(* IEC 61131-3 sources: plc-home-automation/home_automation/lighting_heating_updated/src/lighting, 3 files *)

(* ---- LightingGlobals.st ---- *)
VAR_GLOBAL CONSTANT

    C_DOWNSTAIRS_BATH_MAJOR_LIGHTS_INDEX      : INT := 0;
    C_DOWNSTAIRS_BATH_SHOWER_LIGHTS_INDEX     : INT := 1;
    C_UPSTAIRS_BATH_MAJOR_LIGHTS_INDEX        : INT := 2;
    C_UPSTAIRS_WC_LIGHTS_INDEX                : INT := 3;
    C_UPSTAIRS_BATH_SHOWER_LIGHTS_INDEX       : INT := 4;
    C_HALLWAY_LIGHTS_INDEX                    : INT := 5;
    C_OUTDOOR_LIGHTS_INDEX                    : INT := 6;
    C_HALL_LIGHTS_INDEX                       : INT := 7;
    C_GARAGE_LIGHTS_INDEX                     : INT := 8;
    C_BOILER_LIGHTS_INDEX                     : INT := 9;
    C_MAJOR_STORAGE_LIGHTS_INDEX              : INT := 10;
    C_MINOR_STORAGE_LIGHTS_INDEX              : INT := 11;
    C_GARDEN_BALCONY_LIGHTS_INDEX             : INT := 12;
    C_CHILDRENS_ROOM_2_LIGHTS_INDEX           : INT := 13;
    C_CHILDRENS_ROOM_1_OUTER_LIGHTS_INDEX     : INT := 14;
    C_CHILDRENS_ROOM_1_INNER_LIGHTS_INDEX     : INT := 15;
    C_CHILDRENS_ROOM_3_LIGHTS_INDEX           : INT := 16;
    C_GATE_BALCONY_LIGHTS_INDEX               : INT := 17;
    C_DOWNSTAIRS_BEDROOM_LIGHTS_INDEX         : INT := 18;
    C_KITCHEN_LIGHTS_INDEX                    : INT := 19;
    C_DINING_ROOM_LIGHTS_INDEX                : INT := 20;
    C_LIVING_ROOM_LIGHTS_INDEX                : INT := 21;
    C_TERRACE_LIGHTS_INDEX                    : INT := 22;
//    C_STAIRS_LIGHTS_INDEX               : INT := 23;

    C_LIGHTS_ZONES_COUNT                      : INT := 23;

END_VAR

VAR_GLOBAL

    LIGHTS_INPUTS : ARRAY [0 .. C_LIGHTS_ZONES_COUNT - 1] OF PTR_TO BOOL;
    VIRTUAL_LIGHTS_INPUTS : ARRAY [0 .. C_LIGHTS_ZONES_COUNT - 1] OF PTR_TO BOOL;
    LIGHTS_OUTPUTS : ARRAY [0 .. C_LIGHTS_ZONES_COUNT - 1] OF PTR_TO BOOL;
    LIGHTS_NAMES     : ARRAY [0 .. C_LIGHTS_ZONES_COUNT - 1] OF STRING;

    HALLWAY_LIGHTS_COMBINED_IN : BOOL                      := FALSE;

    VIRTUAL_DOWNSTAIRS_BATH_MAJOR_LIGHTS_IN : BOOL         := FALSE;
    VIRTUAL_DOWNSTAIRS_BATH_SHOWER_LIGHTS_IN : BOOL        := FALSE;
    VIRTUAL_UPSTAIRS_BATH_MAJOR_LIGHTS_IN : BOOL           := FALSE;
    VIRTUAL_UPSTAIRS_WC_LIGHTS_IN : BOOL                   := FALSE;
    VIRTUAL_UPSTAIRS_BATH_SHOWER_LIGHTS_IN : BOOL          := FALSE;
    VIRTUAL_OUTDOOR_LIGHTS_IN : BOOL                       := FALSE;
    VIRTUAL_HALL_LIGHTS_IN : BOOL                          := FALSE;
    VIRTUAL_GARAGE_LIGHTS_IN : BOOL                        := FALSE;
    VIRTUAL_MAJOR_STORAGE_LIGHTS_IN : BOOL                 := FALSE;
    VIRTUAL_MINOR_STORAGE_LIGHTS_IN : BOOL                 := FALSE;
    VIRTUAL_GARDEN_BALCONY_LIGHTS_IN : BOOL                := FALSE;
    VIRTUAL_CHILDRENS_ROOM_2_LIGHTS_IN : BOOL              := FALSE;
    VIRTUAL_CHILDRENS_ROOM_1_OUTER_LIGHTS_IN : BOOL        := FALSE;
    VIRTUAL_CHILDRENS_ROOM_1_INNER_LIGHTS_IN : BOOL        := FALSE;
    VIRTUAL_CHILDRENS_ROOM_3_LIGHTS_IN : BOOL              := FALSE;
    VIRTUAL_GATE_BALCONY_LIGHTS_IN : BOOL                  := FALSE;
    VIRTUAL_DOWNSTAIRS_BEDROOM_LIGHTS_IN : BOOL            := FALSE;
    VIRTUAL_KITCHEN_LIGHTS_IN : BOOL                       := FALSE;
    VIRTUAL_DINING_ROOM_LIGHTS_IN : BOOL                   := FALSE;
    VIRTUAL_LIVING_ROOM_LIGHTS_IN : BOOL                   := FALSE;
    VIRTUAL_TERRACE_LIGHTS_IN : BOOL                       := FALSE;
    VIRTUAL_HALLWAY_LIGHTS_IN : BOOL                       := FALSE;
    VIRTUAL_BOILER_LIGHTS_IN : BOOL                        := FALSE;
//    VIRTUAL_STAIRS_LIGHTS_IN : BOOL                       := FALSE;

    VIRTUAL_EXHAUST_FAN_IN : BOOL                    := FALSE;
    VIRTUAL_CIRCULATION_SWITCH_IN : BOOL             := FALSE;
    VIRTUAL_GARAGE_DOOR_OPENER       : BOOL          := FALSE;

END_VAR

(* ---- Lighting.st ---- *)
// Helper function block
TYPE
  ControllerArray : ARRAY [0 .. C_LIGHTS_ZONES_COUNT - 1] OF ChangeOnOff;
END_TYPE

FUNCTION_BLOCK TurnOffLightsHelper
  VAR_INPUT
    offSignal : BOOL R_EDGE;
  END_VAR

  VAR_IN_OUT
    controllers : ControllerArray;
  END_VAR

  VAR
    i : INT := 0;
  END_VAR

  IF (offSignal) THEN
    FOR i := 0 TO C_LIGHTS_ZONES_COUNT - 1 DO
      controllers[i](requestOff := offSignal);
    END_FOR;
  END_IF;

END_FUNCTION_BLOCK // Helper function block

Program LightingControl

  VAR
    domesticHotWaterCirculation_in : OnThenOffPulse;
    garageGate_in : OnThenOffPulse;

    exhaustRequest     : BOOL := false;
    wcExhaustDelay     : TON;
    wcExhaustDelayTime : TIME := T#4m;
    upstairsBathroomExhaustDelay     : TON;
    upstairsBathroomExhaustDelayTime : TIME := T#8m;
    upstairsShowerExhaustDelay       : TON;
    upstairsShowerExhaustDelayTime   : TIME := T#3m;
    exhaustFan_in     : BathroomFanOnOff;
    exhaustFanRuntime : TIME := T#10m;

    lightsSwitches : ControllerArray;
    lightsControlBasedOnOccupancy : TurnOffLightsHelper;

    i : INT := 0;

  END_VAR

    KITCHEN_FURNITURE_LIGHTS_OUT := TRUE; // We have the door bell in that socket for now.

    domesticHotWaterCirculation_in(
        timeOn := T#2m,
        timeOff := T#20m,
        onSignal := (KERINTGETES_SWITCH_IN OR KITCHEN_FURNITURE_LIGHTS_IN OR VIRTUAL_CIRCULATION_SWITCH_IN),
        name := 'Domestic hot water circulation');
    BOILER_PUMP_PLUG_RIGHT := domesticHotWaterCirculation_in.active;
    VIRTUAL_CIRCULATION_SWITCH_IN := FALSE;

    wcExhaustDelay(IN := UPSTAIRS_WC_LIGHTS_OUT, PT := wcExhaustDelayTime);
    upstairsBathroomExhaustDelay(IN := UPSTAIRS_BATH_MAJOR_LIGHTS_OUT, PT := upstairsBathroomExhaustDelayTime);
    upstairsShowerExhaustDelay(IN := UPSTAIRS_BATH_SHOWER_LIGHTS_OUT, PT := upstairsShowerExhaustDelayTime);
    // No longer needed since we have a full house ventillation system
    // exhaustRequest := wcExhaustDelay.Q OR upstairsBathroomExhaustDelay.Q OR upstairsShowerExhaustDelay.Q;
    exhaustRequest := FALSE;
    exhaustFan_in(timeOn := exhaustFanRuntime, feedOn := exhaustRequest, feedOff := NOT exhaustRequest, change := EXHAUST_FAN_IN OR VIRTUAL_EXHAUST_FAN_IN, name := 'Elszivo ventillator');
    EXHAUST_FAN_OUT := exhaustFan_in.out;
    VIRTUAL_EXHAUST_FAN_IN := FALSE;

    garageGate_in(onSignal := GARAGE_GATE_IN OR VIRTUAL_GARAGE_DOOR_OPENER, timeOn := T#0.2s, timeOff := T#0.2s, name := 'Garage gate');
    GARAGE_GATE_OUT := garageGate_in.active;
    VIRTUAL_GARAGE_DOOR_OPENER := FALSE;

    HALLWAY_LIGHTS_COMBINED_IN := HALLWAY_LIGHTS_IN OR STAIRS_LIGHTS_IN;

    FOR i := 0 TO C_LIGHTS_ZONES_COUNT - 1 DO
        lightsSwitches[i].name := LIGHTS_NAMES[i];
        lightsSwitches[i].requestChange := LIGHTS_INPUTS[i]^ OR VIRTUAL_LIGHTS_INPUTS[i]^;
        lightsSwitches[i]();
        LIGHTS_OUTPUTS[i]^ := lightsSwitches[i].output;
        VIRTUAL_LIGHTS_INPUTS[i]^ := FALSE;
    END_FOR;

    lightsControlBasedOnOccupancy( offSignal := (ALARM_ACTIVE AND GONE_FOR_SHORT_TIME), controllers := lightsSwitches );

END_PROGRAM

(* ---- LightingInit.st ---- *)
PROGRAM LightingInit

    VAR
        initialised : BOOL := false;
    END_VAR;

    IF initialised = FALSE THEN
        initialised := TRUE;

        LIGHTS_INPUTS[C_DOWNSTAIRS_BATH_MAJOR_LIGHTS_INDEX]       := ADR(DOWNSTAIRS_BATH_MAJOR_LIGHTS_IN);
        LIGHTS_INPUTS[C_DOWNSTAIRS_BATH_SHOWER_LIGHTS_INDEX]      := ADR(DOWNSTAIRS_BATH_SHOWER_LIGHTS_IN);
        LIGHTS_INPUTS[C_UPSTAIRS_BATH_MAJOR_LIGHTS_INDEX]         := ADR(UPSTAIRS_BATH_MAJOR_LIGHTS_IN);
        LIGHTS_INPUTS[C_UPSTAIRS_WC_LIGHTS_INDEX]                 := ADR(UPSTAIRS_WC_VIALGITAS_IN);
        LIGHTS_INPUTS[C_UPSTAIRS_BATH_SHOWER_LIGHTS_INDEX]        := ADR(UPSTAIRS_BATH_SHOWER_LIGHTS_IN);
        LIGHTS_INPUTS[C_OUTDOOR_LIGHTS_INDEX]                     := ADR(OUTDOOR_LIGHTS_IN);
        LIGHTS_INPUTS[C_HALL_LIGHTS_INDEX]                        := ADR(HALL_LIGHTS_IN);
        LIGHTS_INPUTS[C_GARAGE_LIGHTS_INDEX]                      := ADR(GARAGE_LIGHTS_IN);
        LIGHTS_INPUTS[C_MAJOR_STORAGE_LIGHTS_INDEX]               := ADR(MAJOR_STORAGE_LIGHTS_IN);
        LIGHTS_INPUTS[C_MINOR_STORAGE_LIGHTS_INDEX]               := ADR(MINOR_STORAGE_LIGHTS_IN);
        LIGHTS_INPUTS[C_GARDEN_BALCONY_LIGHTS_INDEX]              := ADR(GARDEN_BALCONY_LIGHTS_IN);
        LIGHTS_INPUTS[C_CHILDRENS_ROOM_2_LIGHTS_INDEX]            := ADR(CHILDRENS_ROOM_2_LIGHTS_IN);
        LIGHTS_INPUTS[C_CHILDRENS_ROOM_1_OUTER_LIGHTS_INDEX]      := ADR(CHILDRENS_ROOM_1_OUTER_LIGHTS_IN);
        LIGHTS_INPUTS[C_CHILDRENS_ROOM_1_INNER_LIGHTS_INDEX]      := ADR(CHILDRENS_ROOM_1_INNER_LIGHTS_IN);
        LIGHTS_INPUTS[C_CHILDRENS_ROOM_3_LIGHTS_INDEX]            := ADR(CHILDRENS_ROOM_3_LIGHTS_IN);
        LIGHTS_INPUTS[C_GATE_BALCONY_LIGHTS_INDEX]                := ADR(GATE_BALCONY_LIGHTS_IN);
        LIGHTS_INPUTS[C_DOWNSTAIRS_BEDROOM_LIGHTS_INDEX]          := ADR(DOWNSTAIRS_BEDROOM_LIGHTS_IN);
        LIGHTS_INPUTS[C_KITCHEN_LIGHTS_INDEX]                     := ADR(KITCHEN_LIGHTS_IN);
        LIGHTS_INPUTS[C_DINING_ROOM_LIGHTS_INDEX]                 := ADR(DINING_ROOM_LIGHTS_IN);
        LIGHTS_INPUTS[C_LIVING_ROOM_LIGHTS_INDEX]                 := ADR(LIVING_ROOM_LIGHTS_IN);
        LIGHTS_INPUTS[C_TERRACE_LIGHTS_INDEX]                     := ADR(TERRACE_LIGHTS_IN);
        LIGHTS_INPUTS[C_HALLWAY_LIGHTS_INDEX]                     := ADR(HALLWAY_LIGHTS_COMBINED_IN);
        LIGHTS_INPUTS[C_BOILER_LIGHTS_INDEX]                      := ADR(BOILER_LIGHTS_IN);
//        LIGHTS_INPUTS[C_STAIRS_LIGHTS_INDEX]                    := ADR(STAIRS_LIGHTS_IN);

        LIGHTS_OUTPUTS[C_DOWNSTAIRS_BATH_MAJOR_LIGHTS_INDEX]      := ADR(DOWNSTAIRS_BATH_MAJOR_LIGHTS_OUT);
        LIGHTS_OUTPUTS[C_DOWNSTAIRS_BATH_SHOWER_LIGHTS_INDEX]     := ADR(DOWNSTAIRS_BATH_SHOWER_LIGHTS_OUT);
        LIGHTS_OUTPUTS[C_UPSTAIRS_BATH_MAJOR_LIGHTS_INDEX]        := ADR(UPSTAIRS_BATH_MAJOR_LIGHTS_OUT);
        LIGHTS_OUTPUTS[C_UPSTAIRS_WC_LIGHTS_INDEX]                := ADR(UPSTAIRS_WC_LIGHTS_OUT);
        LIGHTS_OUTPUTS[C_UPSTAIRS_BATH_SHOWER_LIGHTS_INDEX]       := ADR(UPSTAIRS_BATH_SHOWER_LIGHTS_OUT);
        LIGHTS_OUTPUTS[C_OUTDOOR_LIGHTS_INDEX]                    := ADR(OUTDOOR_LIGHTS_OUT);
        LIGHTS_OUTPUTS[C_HALL_LIGHTS_INDEX]                       := ADR(HALL_LIGHTS_OUT);
        LIGHTS_OUTPUTS[C_GARAGE_LIGHTS_INDEX]                     := ADR(GARAGE_LIGHTS_OUT);
        LIGHTS_OUTPUTS[C_MAJOR_STORAGE_LIGHTS_INDEX]              := ADR(MAJOR_STORAGE_LIGHTS_OUT);
        LIGHTS_OUTPUTS[C_MINOR_STORAGE_LIGHTS_INDEX]              := ADR(MINOR_STORAGE_LIGHTS_OUT);
        LIGHTS_OUTPUTS[C_GARDEN_BALCONY_LIGHTS_INDEX]             := ADR(GARDEN_BALCONY_LIGHTS_OUT);
        LIGHTS_OUTPUTS[C_CHILDRENS_ROOM_2_LIGHTS_INDEX]           := ADR(CHILDRENS_ROOM_2_LIGHTS_OUT);
        LIGHTS_OUTPUTS[C_CHILDRENS_ROOM_1_OUTER_LIGHTS_INDEX]     := ADR(CHILDRENS_ROOM_1_OUTER_LIGHTS_OUT);
        LIGHTS_OUTPUTS[C_CHILDRENS_ROOM_1_INNER_LIGHTS_INDEX]     := ADR(CHILDRENS_ROOM_1_INNER_LIGHTS_OUT);
        LIGHTS_OUTPUTS[C_CHILDRENS_ROOM_3_LIGHTS_INDEX]           := ADR(CHILDRENS_ROOM_3_LIGHTS_OUT);
        LIGHTS_OUTPUTS[C_GATE_BALCONY_LIGHTS_INDEX]               := ADR(GATE_BALCONY_LIGHTS_OUT);
        LIGHTS_OUTPUTS[C_DOWNSTAIRS_BEDROOM_LIGHTS_INDEX]         := ADR(DOWNSTAIRS_BEDROOM_LIGHTS_OUT);
        LIGHTS_OUTPUTS[C_KITCHEN_LIGHTS_INDEX]                    := ADR(KITCHEN_LIGHTS_OUT);
        LIGHTS_OUTPUTS[C_DINING_ROOM_LIGHTS_INDEX]                := ADR(DINING_ROOM_LIGHTS_OUT);
        LIGHTS_OUTPUTS[C_LIVING_ROOM_LIGHTS_INDEX]                := ADR(LIVING_ROOM_LIGHTS_OUT);
        LIGHTS_OUTPUTS[C_TERRACE_LIGHTS_INDEX]                    := ADR(TERRACE_LIGHTS_OUT);
        LIGHTS_OUTPUTS[C_HALLWAY_LIGHTS_INDEX]                    := ADR(HALLWAY_LIGHTS_OUT);
        LIGHTS_OUTPUTS[C_BOILER_LIGHTS_INDEX]                     := ADR(BOILER_LIGHTS_OUT);
//        LIGHTS_OUTPUTS[C_STAIRS_LIGHTS_INDEX]                   := ADR(HALLWAY_LIGHTS_OUT);

        LIGHTS_NAMES[C_DOWNSTAIRS_BATH_MAJOR_LIGHTS_INDEX]             := 'DOWNSTAIRS_BATH_MAJOR_LIGHTS';
        LIGHTS_NAMES[C_DOWNSTAIRS_BATH_SHOWER_LIGHTS_INDEX]            := 'DOWNSTAIRS_BATH_SHOWER_LIGHTS';
        LIGHTS_NAMES[C_UPSTAIRS_BATH_MAJOR_LIGHTS_INDEX]               := 'UPSTAIRS_BATH_MAJOR_LIGHTS';
        LIGHTS_NAMES[C_UPSTAIRS_WC_LIGHTS_INDEX]                       := 'UPSTAIRS_WC_LIGHTS';
        LIGHTS_NAMES[C_UPSTAIRS_BATH_SHOWER_LIGHTS_INDEX]              := 'UPSTAIRS_BATH_SHOWER_LIGHTS';
        LIGHTS_NAMES[C_OUTDOOR_LIGHTS_INDEX]                           := 'OUTDOOR_LIGHTS';
        LIGHTS_NAMES[C_HALL_LIGHTS_INDEX]                              := 'HALL_LIGHTS';
        LIGHTS_NAMES[C_GARAGE_LIGHTS_INDEX]                            := 'GARAGE_LIGHTS';
        LIGHTS_NAMES[C_MAJOR_STORAGE_LIGHTS_INDEX]                     := 'MAJOR_STORAGE_LIGHTS';
        LIGHTS_NAMES[C_MINOR_STORAGE_LIGHTS_INDEX]                     := 'MINOR_STORAGE_LIGHTS';
        LIGHTS_NAMES[C_GARDEN_BALCONY_LIGHTS_INDEX]                    := 'GARDEN_BALCONY_LIGHTS';
        LIGHTS_NAMES[C_CHILDRENS_ROOM_2_LIGHTS_INDEX]                  := 'CHILDRENS_ROOM_2_LIGHTS';
        LIGHTS_NAMES[C_CHILDRENS_ROOM_1_OUTER_LIGHTS_INDEX]            := 'CHILDRENS_ROOM_1_OUTER_LIGHTS';
        LIGHTS_NAMES[C_CHILDRENS_ROOM_1_INNER_LIGHTS_INDEX]            := 'CHILDRENS_ROOM_1_INNER_LIGHTS';
        LIGHTS_NAMES[C_CHILDRENS_ROOM_3_LIGHTS_INDEX]                  := 'CHILDRENS_ROOM_3_LIGHTS';
        LIGHTS_NAMES[C_GATE_BALCONY_LIGHTS_INDEX]                      := 'GATE_BALCONY_LIGHTS';
        LIGHTS_NAMES[C_DOWNSTAIRS_BEDROOM_LIGHTS_INDEX]                := 'DOWNSTAIRS_BEDROOM_LIGHTS';
        LIGHTS_NAMES[C_KITCHEN_LIGHTS_INDEX]                           := 'KITCHEN_LIGHTS';
        LIGHTS_NAMES[C_DINING_ROOM_LIGHTS_INDEX]                       := 'DINING_ROOM_LIGHTS';
        LIGHTS_NAMES[C_LIVING_ROOM_LIGHTS_INDEX]                       := 'LIVING_ROOM_LIGHTS';
        LIGHTS_NAMES[C_TERRACE_LIGHTS_INDEX]                           := 'TERRACE_LIGHTS';
        LIGHTS_NAMES[C_HALLWAY_LIGHTS_INDEX]                           := 'HALLWAY_LIGHTS';
        LIGHTS_NAMES[C_BOILER_LIGHTS_INDEX]                            := 'BOILER_LIGHTS';
//        LIGHTS_NAMES[C_STAIRS_LIGHTS_INDEX]                          := 'STAIRS_LIGHTS_DOWNSTAIRS';

        VIRTUAL_LIGHTS_INPUTS[C_DOWNSTAIRS_BATH_MAJOR_LIGHTS_INDEX]     := ADR(VIRTUAL_DOWNSTAIRS_BATH_MAJOR_LIGHTS_IN);
        VIRTUAL_LIGHTS_INPUTS[C_DOWNSTAIRS_BATH_SHOWER_LIGHTS_INDEX]    := ADR(VIRTUAL_DOWNSTAIRS_BATH_SHOWER_LIGHTS_IN);
        VIRTUAL_LIGHTS_INPUTS[C_UPSTAIRS_BATH_MAJOR_LIGHTS_INDEX]       := ADR(VIRTUAL_UPSTAIRS_BATH_MAJOR_LIGHTS_IN);
        VIRTUAL_LIGHTS_INPUTS[C_UPSTAIRS_WC_LIGHTS_INDEX]               := ADR(VIRTUAL_UPSTAIRS_WC_LIGHTS_IN);
        VIRTUAL_LIGHTS_INPUTS[C_UPSTAIRS_BATH_SHOWER_LIGHTS_INDEX]      := ADR(VIRTUAL_UPSTAIRS_BATH_SHOWER_LIGHTS_IN);
        VIRTUAL_LIGHTS_INPUTS[C_OUTDOOR_LIGHTS_INDEX]                   := ADR(VIRTUAL_OUTDOOR_LIGHTS_IN);
        VIRTUAL_LIGHTS_INPUTS[C_HALL_LIGHTS_INDEX]                      := ADR(VIRTUAL_HALL_LIGHTS_IN);
        VIRTUAL_LIGHTS_INPUTS[C_GARAGE_LIGHTS_INDEX]                    := ADR(VIRTUAL_GARAGE_LIGHTS_IN);
        VIRTUAL_LIGHTS_INPUTS[C_MAJOR_STORAGE_LIGHTS_INDEX]             := ADR(VIRTUAL_MAJOR_STORAGE_LIGHTS_IN);
        VIRTUAL_LIGHTS_INPUTS[C_MINOR_STORAGE_LIGHTS_INDEX]             := ADR(VIRTUAL_MINOR_STORAGE_LIGHTS_IN);
        VIRTUAL_LIGHTS_INPUTS[C_GARDEN_BALCONY_LIGHTS_INDEX]            := ADR(VIRTUAL_GARDEN_BALCONY_LIGHTS_IN);
        VIRTUAL_LIGHTS_INPUTS[C_CHILDRENS_ROOM_2_LIGHTS_INDEX]          := ADR(VIRTUAL_CHILDRENS_ROOM_2_LIGHTS_IN);
        VIRTUAL_LIGHTS_INPUTS[C_CHILDRENS_ROOM_1_OUTER_LIGHTS_INDEX]    := ADR(VIRTUAL_CHILDRENS_ROOM_1_OUTER_LIGHTS_IN);
        VIRTUAL_LIGHTS_INPUTS[C_CHILDRENS_ROOM_1_INNER_LIGHTS_INDEX]    := ADR(VIRTUAL_CHILDRENS_ROOM_1_INNER_LIGHTS_IN);
        VIRTUAL_LIGHTS_INPUTS[C_CHILDRENS_ROOM_3_LIGHTS_INDEX]          := ADR(VIRTUAL_CHILDRENS_ROOM_3_LIGHTS_IN);
        VIRTUAL_LIGHTS_INPUTS[C_GATE_BALCONY_LIGHTS_INDEX]              := ADR(VIRTUAL_GATE_BALCONY_LIGHTS_IN);
        VIRTUAL_LIGHTS_INPUTS[C_DOWNSTAIRS_BEDROOM_LIGHTS_INDEX]        := ADR(VIRTUAL_DOWNSTAIRS_BEDROOM_LIGHTS_IN);
        VIRTUAL_LIGHTS_INPUTS[C_KITCHEN_LIGHTS_INDEX]                   := ADR(VIRTUAL_KITCHEN_LIGHTS_IN);
        VIRTUAL_LIGHTS_INPUTS[C_DINING_ROOM_LIGHTS_INDEX]               := ADR(VIRTUAL_DINING_ROOM_LIGHTS_IN);
        VIRTUAL_LIGHTS_INPUTS[C_LIVING_ROOM_LIGHTS_INDEX]               := ADR(VIRTUAL_LIVING_ROOM_LIGHTS_IN);
        VIRTUAL_LIGHTS_INPUTS[C_TERRACE_LIGHTS_INDEX]                   := ADR(VIRTUAL_TERRACE_LIGHTS_IN);
        VIRTUAL_LIGHTS_INPUTS[C_HALLWAY_LIGHTS_INDEX]                   := ADR(VIRTUAL_HALLWAY_LIGHTS_IN);
        VIRTUAL_LIGHTS_INPUTS[C_BOILER_LIGHTS_INDEX]                    := ADR(VIRTUAL_BOILER_LIGHTS_IN);
//        VIRTUAL_LIGHTS_INPUTS[C_STAIRS_LIGHTS_INDEX]                  := ADR(VIRTUAL_STAIRS_LIGHTS_IN);
    ELSE
        // No operation
    END_IF;

END_PROGRAM
